// TIA Portal V20 export
TYPE "LER_typeCommunicationControlNode"
// stored: Access Published
   STRUCT
      commands : "LER_typeCommunicationCommands";
      monitoring { S7_SetPoint := 'True'} : "LER_typeCommunicationMonitoring";
   END_STRUCT;
END_TYPE
